FUNCTION cycle_Logger : BOOL
VAR_INPUT
	pLogger			: POINTER TO T_LoggerSendData;
END_VAR
VAR
END_VAR

(* Copyright 2017 Cimpress

Licensed under the Apache License, Version 2.0 (the "License");
you may not use this file except in compliance with the License.
You may obtain a copy of the License at

http://www.apache.org/licenses/LICENSE-2.0

Unless required by applicable law or agreed to in writing, software
distributed under the License is distributed on an "AS IS" BASIS,
WITHOUT WARRANTIES OR CONDITIONS OF ANY KIND, either express or implied.
See the License for the specific language governing permissions and
limitations under the License. *)

pLogger^.fbFifo();

END_FUNCTION

(* stored: Version 1.1.0.1, ProductVersion 3.1.4019.2
   POU cycle_Logger: Id {12d75f6a-b747-419a-858a-a56959f7e0d5}, SpecialFunc None *)
